// TwinCAT 3 PLC project TcTest
// Title: TcTest
// Company: Test company
// Author: Unknown
// ProjectVersion: 0.0.0.1
// Description: Test code for testing purposes.
// ProgramVersion: 3.1.4026.9
// libraries:
//   Tc2_Standard, * (Beckhoff Automation GmbH)
//   Tc2_System, * (Beckhoff Automation GmbH)
//   Tc3_MiniFrame, * (Gayfiles)
// project tree:
//   / PlcTask.TcTTO
//   POUs/ E_OffOnTest.TcDUT, FB_Aggregate.TcPOU (not stored), FB_TestDevice.TcPOU (not stored), MAIN.TcPOU (not stored)
//   Version/ Global_Version.TcGVL
// real-time tasks:
//   TASK PlcTask: cycle T#10ms, priority 20, ADS port 350

CONFIGURATION TcTest
    RESOURCE PLC ON TwinCAT3
        TASK PlcTask(INTERVAL := T#10ms, PRIORITY := 20);
        PROGRAM MAIN WITH PlcTask : MAIN;
    END_RESOURCE
END_CONFIGURATION

// ---- POUs/E_OffOnTest.TcDUT
{attribute 'qualified_only'}
TYPE E_OffOnTest :
(
	_invalid := 0,
	
	Auto := 1,
	Off := 2,
	On := 3
) UDINT;
END_TYPE

// ---- Version/Global_Version.TcGVL
{attribute 'TcGenerated'}
{attribute 'no-analysis'}
{attribute 'linkalways'}
// This function has been automatically generated from the project information.
VAR_GLOBAL CONSTANT
	{attribute 'const_non_replaced'}
	stLibVersion_TcTest : ST_LibVersion := (iMajor := 0, iMinor := 0, iBuild := 0, iRevision := 1, nFlags := 0, sVersion := '0.0.0.1');
END_VAR
